FUNCTION_BLOCK MoveModuloMoverToPosition  IMPLEMENTS I_Task, I_Cyclic, I_Object, I_Abortable
VAR
	moveAbs	: MC_MoveAbsoluteCA;
	_Axis : REFERENCE TO AXIS_REF;
	_stOptions : ST_MoveAbsoluteCAOptions;
END_VAR

{analysis -2}

METHOD Abort : BOOL
moveAbs.Execute := FALSE;
moveAbs.Position := moveAbs.Velocity := 0;
_MoveMover := false;
_Busy := FALSE;
Abort := true;
State := 0;
END_METHOD

PROPERTY PUBLIC Acceleration : mc_lreal
GET
Acceleration := moveAbs.Acceleration;
END_GET
SET
moveAbs.Acceleration := Acceleration;
END_SET
END_PROPERTY

PROPERTY AxisRef : reference to Axis_ref
GET
AxisRef	REF= _Axis;
END_GET
SET
_Axis REF= AxisRef;
END_SET
END_PROPERTY

PROPERTY Busy : BOOL
GET
Busy := moveAbs.Busy;
END_GET
END_PROPERTY

METHOD Cycle : HRESULT
VAR_INPUT
END_VAR
moveAbs(Axis := _Axis, Options := _stOptions);
moveAbs.Execute := false;
END_METHOD

PROPERTY PUBLIC Deceleration : mc_lreal
GET
Deceleration := moveAbs.Deceleration;
END_GET
SET
moveAbs.Deceleration := Deceleration;
END_SET
END_PROPERTY

PROPERTY Done : BOOL
GET
Done := moveAbs.Done;
END_GET
END_PROPERTY

PROPERTY Error : BOOL
GET
Error := moveAbs.Error;
END_GET
END_PROPERTY

PROPERTY PUBLIC Gap : mc_lreal
GET
Gap := moveAbs.Gap;
END_GET
SET
moveAbs.Gap := Gap;
END_SET
END_PROPERTY

PROPERTY PUBLIC Jerk : mc_lreal
GET
Jerk := moveAbs.Jerk;
END_GET
SET
moveAbs.Jerk := Jerk;
END_SET
END_PROPERTY

METHOD MoveTo : BOOL
VAR_INPUT
	Position : MC_LREAL;
	Velocity : MC_LREAL;
	Direction: Tc3_Mc3Definitions.MC_DIRECTION;
	Turns: UDINT;
END_VAR
moveAbs.Position := Position;
moveAbs.Velocity := Velocity;
moveAbs.Direction := Direction;
moveAbs.Options.AdditionalTurns := Turns;
moveAbs.Execute := MoveTo := TRUE;
END_METHOD

PROPERTY PUBLIC Options : ST_MoveAbsoluteCAOptions
GET
Options := _stOptions;
END_GET
SET
_stOptions := Options;
END_SET
END_PROPERTY

METHOD RegisterWithParent
VAR_INPUT
	Runner	: Base_Library.I_HostObjects;
END_VAR
Runner.RegisterCyclic(THIS^);
Runner.RegisterAbortable(THIS^);
Runner.RegisterTask(THIS^);
END_METHOD

END_FUNCTION_BLOCK

(* stored: Version 1.1.0.1
   POU MoveModuloMoverToPosition: Id {86a89fc0-d952-4342-8bc4-3e7afaf8d6b0}, SpecialFunc None
   Method Abort: Id {5c5502fe-cfbb-4721-939d-6b8391fd3812}
   Property Acceleration: Id {bd8e2346-8872-4feb-ac95-f472cf2ca2c7}
   Get Get: Id {c4ef743d-06c1-4445-9890-b82ffba396f1}
   Set Set: Id {1c8827c9-2f8f-4b77-8024-4b0046d69ac2}
   Property AxisRef: Id {f580a694-3b65-4030-87ca-bcac6820ed0e}
   Get Get: Id {7844fea5-7585-46ce-89d1-d518d3791463}
   Set Set: Id {8364ed17-5c2f-4208-b144-b38ccd52dc0b}
   Property Busy: Id {98ae5732-f508-463a-8f9c-9f54ad1821f5}
   Get Get: Id {84ba2f1a-36fd-4d7b-97cb-ca57f0f3f0c7}
   Method Cycle: Id {4cb00213-de2b-40d2-a495-86e25cb3d039}
   Property Deceleration: Id {9b084d4a-e02d-4702-912a-4bc5910ddae2}
   Get Get: Id {a47d2d08-c000-41b9-a1f9-a582ebe1b9d1}
   Set Set: Id {82a7f264-1036-48b4-a621-2fa4d8fd0895}
   Property Done: Id {706feeb3-2a28-4a2a-b819-7bb55bd73ff5}
   Get Get: Id {37c3e926-1b46-4356-8064-b4a1dfbf3ce5}
   Property Error: Id {d69fd401-b2dd-44f6-914b-954c635c1b05}
   Get Get: Id {c20a1bf9-e383-400a-99fa-a6607965fe21}
   Property Gap: Id {6f40f3be-1ac5-4f41-a512-900c33b72e2e}
   Get Get: Id {d520ecb2-c250-4598-84bd-dc6b0a2aef6c}
   Set Set: Id {49d06445-a9cb-4b50-a172-a728c79a3bc7}
   Property Jerk: Id {557e6884-85fe-4a0b-9fbe-e021e4eb6165}
   Get Get: Id {43424688-9bf6-468e-9d81-7307bd08e1b7}
   Set Set: Id {fbdecc92-c967-41e0-99c8-b2c9f3bf8bd0}
   Method MoveTo: Id {42a523a0-ad8a-4fac-a76b-d1875ec2f808}
   Property Options: Id {1dd7fc51-dd5a-4f57-a3ca-696f6637a39e}
   Get Get: Id {179a8440-f33d-4396-9725-56d6b0191700}
   Set Set: Id {18307288-77cd-4621-a1f2-e62bd90c9ccf}
   Method RegisterWithParent: Id {d5091b4b-bfac-4bc2-8672-2fc22997a298} *)
